(* IEC 61131-3 sources: AXOpen/src/inspectors/ctrl/src/interfaces, 3 files *)

(* ---- IAxoComprehensiveResult.st ---- *)
USING AXOpen.Core;
NAMESPACE AXOpen.Inspectors
    INTERFACE IAxoComprehensiveResult

        METHOD GetResult : eOverallResult
        END_METHOD

        METHOD GetFailures : STRING
        END_METHOD

        METHOD GetErrorCodes : STRING
        END_METHOD

        METHOD SetResult
            VAR_INPUT
                inResult: eOverallResult;
            END_VAR
        END_METHOD

        METHOD SetFailures
            VAR_INPUT
                inFailures: STRING;
            END_VAR
        END_METHOD

        METHOD SetErrorCodes
            VAR_INPUT
                inErrorCodes: STRING;
            END_VAR
        END_METHOD

        METHOD AddFailure
            VAR_INPUT
                inFailure: STRING;
            END_VAR
        END_METHOD

        METHOD AddErrorCode
            VAR_INPUT
                inErrorCode: STRING;
            END_VAR
        END_METHOD

    END_INTERFACE
END_NAMESPACE

(* ---- IInspector.st ---- *)
USING AXOpen.Core;
NAMESPACE AXOpen.Inspectors
    INTERFACE IInspector

        METHOD Busy : BOOL
        END_METHOD

        METHOD CommonData : REF_TO AxoInspectorData
        END_METHOD

        METHOD Coordinator : IAxoCoordinator
        END_METHOD

        METHOD Done : BOOL
        END_METHOD

        METHOD CheckOverInspection : BOOL
        END_METHOD

        METHOD Result : eInspectorResult
        END_METHOD

        METHOD Dialog : BOOL
            VAR_INPUT
                inRetryStep: IAxoStep;
                inTerminateStep: IAxoStep;
            END_VAR

        END_METHOD

        METHOD  RestoreInspectorTask : BOOL
        END_METHOD

        METHOD OnFail : IOnFail
        END_METHOD

        METHOD UpdateComprehensiveResult : IInspector

            VAR_IN_OUT
                inoResult : AxoComprehensiveResult;
            END_VAR

        END_METHOD

        METHOD Inspect : IInspector
            VAR_INPUT
                inParent : AXOpen.Core.IAxoObject;
                inData : REF_TO AxoAnalogueInspectorData;
                Status : LREAL;
            END_VAR
        END_METHOD

        METHOD Inspect : IInspector
            VAR_INPUT
                inParent : AXOpen.Core.IAxoObject;
                inData : REF_TO AxoDigitalInspectorData;
                Status : BOOL;
            END_VAR
        END_METHOD

        METHOD Inspect : IInspector
            VAR_INPUT
                inParent : AXOpen.Core.IAxoObject;
                inData : REF_TO AxoDataInspectorData;
                Status : STRING;
            END_VAR
        END_METHOD
    END_INTERFACE
END_NAMESPACE

(* ---- IOnFail.st ---- *)
NAMESPACE AXOpen.Inspectors
    INTERFACE IOnFail

        METHOD CarryOn : BOOL
        END_METHOD

        METHOD RetryWithStep : BOOL
            VAR_INPUT
                /// State from which the inspection will restart.
                inRetryStep : AXOpen.Core.IAxoStep;
            END_VAR
        END_METHOD

        METHOD Dialog : BOOL
            VAR_INPUT
                inRetryStep: AXOpen.Core.IAxoStep;
                inTerminateStep: AXOpen.Core.IAxoStep;
            END_VAR
        END_METHOD

        METHOD TerminateWithStep : BOOL
            VAR_INPUT
                /// State from which the inspection will restart.
                inTerminateStep : AXOpen.Core.IAxoStep;
            END_VAR
        END_METHOD

    END_INTERFACE
END_NAMESPACE
